{attribute 'qualified_only'}
VAR_GLOBAL
	//LCP 1 (Bank1 ) Instrument reading
	R2_03 : ST_InstrumentReading;
	//R2_02 : ARRAY [0..7] OF ST_InstrumentReading; // in case we need another card for R2
	R3_04 : ST_InstrumentReading;
	
END_VAR

(* stored: Version 1.1.0.1, ProductVersion 3.1.4024.11
   GVL InstrumentReading: Id {666695df-69ac-4ec1-8d55-e50ecd0788a4} *)
